# B&R Automation Studio project TD52 (part 87)

#### AI50toIT_mdl.h
```c
/********************************************************************
 * COPYRIGHT -- Bernecker + Rainer Industrie-Elektronik Ges.m.b.H.
 ********************************************************************
 * Program: AI50toIT_mdl
 * File: AI50toIT_mdl.h
 * Author: 105055527
 * Created: Thu Sep 11 18:05:22 2014
 ********************************************************************
 * Header for program AI50toIT_mdl
 ********************************************************************
 * Generated with B&R Automation Studio Target for Simulink V4.2
 * (ERT based)
 ********************************************************************/

#ifndef RTW_HEADER_AI50toIT_mdl_h_
#define RTW_HEADER_AI50toIT_mdl_h_
#ifndef AI50toIT_mdl_COMMON_INCLUDES_
# define AI50toIT_mdl_COMMON_INCLUDES_
#include <math.h>
#include "rtwtypes.h"
#endif                                 /* AI50toIT_mdl_COMMON_INCLUDES_ */

#include "AI50toIT_mdl_types.h"
#include "lAI50toIT.h"

/* Macros for accessing real-time model data structure */
#ifndef rtmGetErrorStatus
# define rtmGetErrorStatus(rtm)        ((void*) 0)
#endif

#ifndef rtmSetErrorStatus
# define rtmSetErrorStatus(rtm, val)   ((void) 0)
#endif

#ifndef rtmGetStopRequested
# define rtmGetStopRequested(rtm)      ((void*) 0)
#endif

#ifndef MIN
#define MIN(a,b)                       ((a) < (b) ? (a) : (b))
#endif

#ifndef MAX
#define MAX(a,b)                       ((a) > (b) ? (a) : (b))
#endif

/* Block signals (auto storage) */

/* Block states (auto storage) for system '<Root>' */

/* External inputs (root inport signals with auto storage) */

/* External outputs (root outports fed by signals with auto storage) */

/* Block signals (auto storage) */
extern BlockIO_AI50toIT_mdl AI50toIT_mdl_B;

/* Block states (auto storage) */
extern D_Work_AI50toIT_mdl AI50toIT_mdl_DWork;

/* External inputs (root inport signals with auto storage) */
extern ExternalInputs_AI50toIT_mdl AI50toIT_mdl_U;

/* External outputs (root outports fed by signals with auto storage) */
extern ExternalOutputs_AI50toIT_mdl AI50toIT_mdl_Y;

/* Model entry point functions */
extern void AI50toIT_mdl_initialize(struct AI50toIT* inst);
extern void AI50toIT_mdl_step(struct AI50toIT* inst);
extern void AI50toIT_mdl_terminate(struct AI50toIT* inst);

/*-
 * The generated code includes comments that allow you to trace directly
 * back to the appropriate location in the model.  The basic format
 * is <system>/block_name, where system is the system number (uniquely
 * assigned by Simulink) and block_name is the name of the block.
 *
 * Use the MATLAB hilite_system command to trace the generated code back
 * to the model.  For example,
 *
 * hilite_system('<S3>')    - opens system 3
 * hilite_system('<S3>/Kp') - opens and selects block Kp which resides in S3
 *
 * Here is the system hierarchy for this model
 *
 * '<Root>' : 'AI50toIT_mdl'
 * '<S1>'   : 'AI50toIT_mdl/AI50 filt'
 * '<S2>'   : 'AI50toIT_mdl/DocBlock'
 * '<S3>'   : 'AI50toIT_mdl/Environment Controller'
 * '<S4>'   : 'AI50toIT_mdl/Environment Controller1'
 * '<S5>'   : 'AI50toIT_mdl/Model Info'
 * '<S6>'   : 'AI50toIT_mdl/PID'
 * '<S7>'   : 'AI50toIT_mdl/Saturation Dynamic'
 * '<S8>'   : 'AI50toIT_mdl/PID/PID Autocoding2'
 * '<S9>'   : 'AI50toIT_mdl/PID/Saturation Dynamic'
 * '<S10>'  : 'AI50toIT_mdl/PID/PID Autocoding2/Dead Zone Dynamic'
 * '<S11>'  : 'AI50toIT_mdl/PID/PID Autocoding2/PID'
 * '<S12>'  : 'AI50toIT_mdl/PID/PID Autocoding2/PID/Clamping circuit'
 * '<S13>'  : 'AI50toIT_mdl/PID/PID Autocoding2/PID/Saturation Dynamic'
 * '<S14>'  : 'AI50toIT_mdl/PID/PID Autocoding2/PID/Clamping circuit/Compare To Constant'
 */
#endif                                 /* RTW_HEADER_AI50toIT_mdl_h_ */
```

#### AI50toIT_mdl_private.h
```c
/********************************************************************
 * COPYRIGHT -- Bernecker + Rainer Industrie-Elektronik Ges.m.b.H.
 ********************************************************************
 * Program: AI50toIT_mdl
 * File: AI50toIT_mdl_private.h
 * Author: 105055527
 * Created: Thu Sep 11 18:05:22 2014
 ********************************************************************
 * Header for program AI50toIT_mdl
 ********************************************************************
 * Generated with B&R Automation Studio Target for Simulink V4.2
 * (ERT based)
 ********************************************************************/

#ifndef RTW_HEADER_AI50toIT_mdl_private_h_
#define RTW_HEADER_AI50toIT_mdl_private_h_
#include "rtwtypes.h"
#include <bur/plctypes.h>
#ifndef __RTWTYPES_H__
#error This file requires rtwtypes.h to be included
#else
#ifdef TMWTYPES_PREVIOUSLY_INCLUDED
#error This file requires rtwtypes.h to be included before tmwtypes.h
#else

/* Check for inclusion of an incorrect version of rtwtypes.h */
#ifndef RTWTYPES_ID_C08S16I32L32N32F1
#error This code was generated with a different "rtwtypes.h" than the file included
#endif                                 /* RTWTYPES_ID_C08S16I32L32N32F1 */
#endif                                 /* TMWTYPES_PREVIOUSLY_INCLUDED */
#endif                                 /* __RTWTYPES_H__ */

#ifndef MIN
#define MIN(a,b)                       ((a) < (b) ? (a) : (b))
#endif

#ifndef MAX
#define MAX(a,b)                       ((a) > (b) ? (a) : (b))
#endif

/* Imported (extern) block parameters */
extern real32_T Kt;                    /* Variable: Kt
                                        * Referenced by: '<S6>/Constant10'
                                        */
extern real32_T N;                     /* Variable: N
                                        * Referenced by: '<S6>/Constant8'
                                        */
extern real32_T T_filt_AI50;           /* Variable: T_filt_AI50
                                        * Referenced by: '<S1>/Constant3'
                                        */
extern real32_T deadband;              /* Variable: deadband
                                        * Referenced by: '<S6>/Constant11'
                                        */
extern real32_T kd;                    /* Variable: kd
                                        * Referenced by: '<S6>/Constant7'
                                        */
extern real32_T ki;                    /* Variable: ki
                                        * Referenced by: '<S6>/Constant6'
                                        */
extern real32_T kp;                    /* Variable: kp
                                        * Referenced by: '<S6>/Constant5'
                                        */
extern real32_T umax;                  /* Variable: umax
                                        * Referenced by: '<S6>/Constant16'
                                        */
extern real32_T umin;                  /* Variable: umin
                                        * Referenced by: '<S6>/Constant17'
                                        */
extern int16_T mode;                   /* Variable: mode
                                        * Referenced by: '<S6>/Constant'
                                        */
extern boolean_T invert;               /* Variable: invert
                                        * Referenced by: '<S6>/Constant4'
                                        */
extern boolean_T reset;                /* Variable: reset
                                        * Referenced by:
                                        *   '<S1>/Constant2'
                                        *   '<S6>/Constant1'
                                        */

#endif                                 /* RTW_HEADER_AI50toIT_mdl_private_h_ */
```

#### AI50toIT_mdl_types.h
```c
/********************************************************************
 * COPYRIGHT -- Bernecker + Rainer Industrie-Elektronik Ges.m.b.H.
 ********************************************************************
 * Program: AI50toIT_mdl
 * File: AI50toIT_mdl_types.h
 * Author: 105055527
 * Created: Thu Sep 11 18:05:22 2014
 ********************************************************************
 * Header for program AI50toIT_mdl
 ********************************************************************
 * Generated with B&R Automation Studio Target for Simulink V4.2
 * (ERT based)
 ********************************************************************/

#ifndef RTW_HEADER_AI50toIT_mdl_types_h_
#define RTW_HEADER_AI50toIT_mdl_types_h_
#ifndef MIN
#define MIN(a,b)                       ((a) < (b) ? (a) : (b))
#endif

#ifndef MAX
#define MAX(a,b)                       ((a) > (b) ? (a) : (b))
#endif
#endif                                 /* RTW_HEADER_AI50toIT_mdl_types_h_ */
```

#### rtwtypes.h
```c
/********************************************************************
 * COPYRIGHT -- Bernecker + Rainer Industrie-Elektronik Ges.m.b.H.
 ********************************************************************
 * Program: AI50toIT_mdl
 * File: rtwtypes.h
 * Author: 105055527
 * Created: Thu Sep 11 18:05:22 2014
 ********************************************************************
 * Header for program AI50toIT_mdl
 ********************************************************************
 * Generated with B&R Automation Studio Target for Simulink V4.2
 * (ERT based)
 ********************************************************************/

#ifndef __RTWTYPES_H__
#define __RTWTYPES_H__
#ifndef TRUE
# define TRUE                          (1U)
#endif

#ifndef FALSE
# define FALSE                         (0U)
#endif

#ifndef __TMWTYPES__
#define __TMWTYPES__
#include <limits.h>

/*=======================================================================*
 * Target hardware information
 *   Device type: Intel->x86/Pentium
 *   Number of bits:     char:   8    short:   16    long:  32
 *                       long:  32
 *                       native word size:  32
 *   Byte ordering: LittleEndian
 *   Signed integer division rounds to: Zero
 *   Shift right on a signed integer as arithmetic shift: on
 *=======================================================================*/

/*=======================================================================*
 * Fixed width word size data types:                                     *
 *   int8_T, int16_T, int32_T     - signed 8, 16, or 32 bit integers     *
 *   uint8_T, uint16_T, uint32_T  - unsigned 8, 16, or 32 bit integers   *
 *   real32_T, real64_T           - 32 and 64 bit floating point numbers *
 *=======================================================================*/
typedef signed char int8_T;
typedef unsigned char uint8_T;
typedef short int16_T;
typedef unsigned short uint16_T;
typedef long int32_T;
typedef unsigned long uint32_T;
typedef float real32_T;
typedef double real64_T;

/*===========================================================================*
 * Generic type definitions: real_T, time_T, boolean_T, int_T, uint_T,       *
 *                           ulong_T, char_T and byte_T.                     *
 *===========================================================================*/
typedef double real_T;
typedef double time_T;
typedef unsigned char boolean_T;
typedef long int_T;
typedef unsigned long uint_T;
typedef unsigned long ulong_T;
typedef char char_T;
typedef unsigned char uchar_T;
typedef char_T byte_T;

/*=======================================================================*
 * Min and Max:                                                          *
 *   int8_T, int16_T, int32_T     - signed 8, 16, or 32 bit integers     *
 *   uint8_T, uint16_T, uint32_T  - unsigned 8, 16, or 32 bit integers   *
 *=======================================================================*/
#define MAX_int8_T                     ((int8_T)(127))
#define MIN_int8_T                     ((int8_T)(-128))
#define MAX_uint8_T                    ((uint8_T)(255U))
#define MIN_uint8_T                    ((uint8_T)(0U))
#define MAX_int16_T                    ((int16_T)(32767))
#define MIN_int16_T                    ((int16_T)(-32768))
#define MAX_uint16_T                   ((uint16_T)(65535U))
#define MIN_uint16_T                   ((uint16_T)(0U))
#define MAX_int32_T                    ((int32_T)(2147483647))
#define MIN_int32_T                    ((int32_T)(-2147483647-1))
#define MAX_uint32_T                   ((uint32_T)(0xFFFFFFFFU))
#define MIN_uint32_T                   ((uint32_T)(0U))

/* Logical type definitions */
#if (!defined(__cplusplus)) && (!defined(__true_false_are_keywords))
#  ifndef false
#   define false                       (0U)
#  endif

#  ifndef true
#   define true                        (1U)
#  endif
#endif

/*
 * Simulink Coder assumes the code is compiled on a target using a 2's complement representation
 * for signed integer values.
 */
#if ((SCHAR_MIN + 1) != -SCHAR_MAX)
#error "This code must be compiled using a 2's complement representation for signed integer values"
#endif

/* This ID is used to detect inclusion of an incompatible rtwtypes.h */
#define RTWTYPES_ID_C08S16I32L32N32F1
#else                                  /* __TMWTYPES__ */
#define TMWTYPES_PREVIOUSLY_INCLUDED
#endif                                 /* __TMWTYPES__ */

/* Block D-Work pointer type */
typedef void * pointer_T;

/* Simulink specific types */
#ifndef __SIMSTRUC_TYPES_H__
#define __SIMSTRUC_TYPES_H__

/* Trigger directions: falling, either, and rising */
typedef enum {
  FALLING_ZERO_CROSSING = -1,
  ANY_ZERO_CROSSING = 0,
  RISING_ZERO_CROSSING = 1
} ZCDirection;

/* Previous state of a trigger signal */
typedef uint8_T ZCSigState;

/* Initial value of a trigger zero crossing signal */
#define UNINITIALIZED_ZCSIG            0x03U
#define NEG_ZCSIG                      0x02U
#define POS_ZCSIG                      0x01U
#define ZERO_ZCSIG                     0x00U

/* Current state of a trigger signal */
typedef enum {
  FALLING_ZCEVENT = -1,
  NO_ZCEVENT = 0,
  RISING_ZCEVENT = 1
} ZCEventType;

#endif                                 /* __SIMSTRUC_TYPES_H__ */
#endif                                 /* __RTWTYPES_H__ */

#ifndef MIN
#define MIN(a,b)                       ((a) < (b) ? (a) : (b))
#endif

#ifndef MAX
#define MAX(a,b)                       ((a) > (b) ? (a) : (b))
#endif
```

#### AI50toIT.c
```c
/********************************************************************
 * COPYRIGHT -- Bernecker + Rainer Industrie-Elektronik Ges.m.b.H.
 ********************************************************************
 * Program: AI50toIT_mdl
 * File: AI50toIT.c
 * Author: 105055527
 * Created: Thu Sep 11 18:05:22 2014
 ********************************************************************
 * Implementation of program AI50toIT_mdl
 ********************************************************************
 * Generated with B&R Automation Studio Target for Simulink V4.2
 * (ERT based)
 ********************************************************************/
#include <bur/plctypes.h>
#include "AI50toIT_mdl.h"
#include "rtwtypes.h"

/* Defines */
#define SS_TERMINATE 4
#define SS_OUTPUT 3
#define SS_INITIALIZE 2

/*  Data Types */

/**************************** GLOBAL DATA *************************************/
/*  Definitions */

/*  Declarations  */

/***************************** FILE SCOPE DATA ********************************/

/*************************** FUNCTIONS ****************************************/
#ifdef __cplusplus

unsigned long bur_heap_size = 6553500;

#endif

void AI50toIT(struct AI50toIT* inst)
{

  switch (inst->ssMethodType)
  {
   case SS_INITIALIZE:
    /* call model initialize function */
    AI50toIT_mdl_initialize(inst);
    break;

   case SS_OUTPUT:
    /* call model step function */
    AI50toIT_mdl_step(inst);

    break;

   case SS_TERMINATE:
    /* call model terminate function */
    AI50toIT_mdl_terminate(inst);
    break;
  }
}

/*****************************************************************************
   Function block sample time: 0.08s
 *****************************************************************************/

/*****************************************************************************
   B&R Automation Studio Target for Simulink Version: A4.5.1 (27-Jul-2015)
 *****************************************************************************/

/*======================== TOOL VERSION INFORMATION ==========================*
 * MATLAB 8.0 (R2012b)20-Jul-2012                                             *
 * Simulink 8.0 (R2012b)20-Jul-2012                                           *
 * Simulink Coder 8.3 (R2012b)20-Jul-2012                                     *
 * Embedded Coder 6.3 (R2012b)20-Jul-2012                                     *
 * Stateflow 8.0 (R2012b)20-Jul-2012                                          *
 *============================================================================*/

/*======================= LICENSE IN USE INFORMATION =========================*
 * matlab                                                                     *
 * matlab_coder                                                               *
 * real-time_workshop                                                         *
 * rtw_embedded_coder                                                         *
 * simulink                                                                   *
 *============================================================================*/
```

#### AI50toIT_mdl.c
```c
/********************************************************************
 * COPYRIGHT -- Bernecker + Rainer Industrie-Elektronik Ges.m.b.H.
 ********************************************************************
 * Program: AI50toIT_mdl
 * File: AI50toIT_mdl.c
 * Author: 105055527
 * Created: Thu Sep 11 18:05:22 2014
 ********************************************************************
 * Implementation of program AI50toIT_mdl
 ********************************************************************
 * Generated with B&R Automation Studio Target for Simulink V4.2
 * (ERT based)
 ********************************************************************/
#include "AI50toIT_mdl.h"
#include "AI50toIT_mdl_private.h"

/*  Defines */

/*  Data Types */

/**************************** GLOBAL DATA *************************************/
/*  Definitions */

/* Block signals (auto storage) */
struct BlockIO_AI50toIT_mdl AI50toIT_mdl_B;

/* Block states (auto storage) */
struct D_Work_AI50toIT_mdl AI50toIT_mdl_DWork;

/* External inputs (root inport signals with auto storage) */
ExternalInputs_AI50toIT_mdl AI50toIT_mdl_U;

/* External outputs (root outports fed by signals with auto storage) */
ExternalOutputs_AI50toIT_mdl AI50toIT_mdl_Y;

/*  Declarations  */

/***************************** FILE SCOPE DATA ********************************/

/*************************** FUNCTIONS ****************************************/

/* Model step function */
void AI50toIT_mdl_step(struct AI50toIT* inst)
{
  real32_T rtb_Add[25];
  real32_T rtb_Abs[25];
  real32_T rtb_Trackingswitch;
  real32_T rtb_Invertswitch;
  real32_T rtb_SumI1[25];
  boolean_T rtb_LowerRelop1_k[25];
  int32_T i;
  real32_T rtb_SumI;
  real32_T rtb_SumI_0;

  /* S-Function (bur_in): '<Root>/Input16' */
  {
    int_T i1;
    real32_T *y0 = AI50toIT_mdl_B.Input16;
    for (i1=0; i1 < 25; i1++) {
      y0[i1] = inst->uman[i1];
    }
  }

  /* Switch: '<S8>/Invert switch' incorporates:
   *  Constant: '<S6>/Constant4'
   *  Constant: '<S8>/Constant2'
   *  Constant: '<S8>/Constant3'
   */
  if ((int32_T)inst->invert > 0) {
    rtb_Invertswitch = -1.0F;
  } else {
    rtb_Invertswitch = 1.0F;
  }

  /* End of Switch: '<S8>/Invert switch' */

  /* S-Function (bur_in): '<Root>/Input5' */
  AI50toIT_mdl_B.Input5 = inst->AI50ref;

  /* S-Function (bur_in): '<Root>/Input8' */
  {
    int_T i1;
    real32_T *y0 = AI50toIT_mdl_B.Input8;
    for (i1=0; i1 < 25; i1++) {
      y0[i1] = inst->AI50offset[i1];
    }
  }

  /* S-Function (bur_in): '<Root>/Input3' */
  {
    int_T i1;
    real32_T *y0 = AI50toIT_mdl_B.Input3;
    for (i1=0; i1 < 25; i1++) {
      y0[i1] = inst->AI50offset_knck[i1];
    }
  }

  /* S-Function (bur_in): '<Root>/Input4' */
  AI50toIT_mdl_B.Input4 = inst->K_knck;

  /* Sum: '<Root>/Add' incorporates:
   *  Product: '<Root>/Product'
   */
  for (i = 0; i < 25; i++) {
    rtb_Add[i] = (AI50toIT_mdl_B.Input5 + AI50toIT_mdl_B.Input8[i]) +
      AI50toIT_mdl_B.Input3[i] * AI50toIT_mdl_B.Input4;
  }

  /* End of Sum: '<Root>/Add' */

  /* DiscreteIntegrator: '<S1>/Discrete-Time Integrator' incorporates:
   *  Constant: '<S1>/Constant2'
   */
  if (inst->reset || (AI50toIT_mdl_DWork.DiscreteTimeIntegrator_PrevRese != 0)) {
    for (i = 0; i < 25; i++) {
      AI50toIT_mdl_DWork.DiscreteTimeIntegrator_DSTATE[i] = 10.0F;
    }
  }

  for (i = 0; i < 25; i++) {
    /* DiscreteIntegrator: '<S1>/Discrete-Time Integrator' */
    AI50toIT_mdl_B.DiscreteTimeIntegrator[i] =
      AI50toIT_mdl_DWork.DiscreteTimeIntegrator_DSTATE[i];

    /* Sum: '<S8>/Sum' incorporates:
     *  Product: '<S8>/Product'
     *  Product: '<S8>/Product1'
     */
    rtb_Trackingswitch = rtb_Add[i] - AI50toIT_mdl_B.DiscreteTimeIntegrator[i];

    /* Switch: '<S10>/Switch' incorporates:
     *  Constant: '<S6>/Constant11'
     *  Gain: '<S8>/Gain1'
     *  RelationalOperator: '<S10>/u_GTE_up'
     *  RelationalOperator: '<S10>/u_GT_lo'
     *  Switch: '<S10>/Switch1'
     */
    if (rtb_Trackingswitch >= inst->deadband) {
      rtb_SumI = inst->deadband;
    } else if (rtb_Trackingswitch > -inst->deadband) {
      /* Switch: '<S10>/Switch1' */
      rtb_SumI = rtb_Trackingswitch;
    } else {
      rtb_SumI = -inst->deadband;
    }

    /* End of Switch: '<S10>/Switch' */

    /* Product: '<S8>/Product2' incorporates:
     *  Sum: '<S10>/Diff'
     */
    AI50toIT_mdl_B.Product2[i] = (rtb_Trackingswitch - rtb_SumI) *
      rtb_Invertswitch;

    /* Product: '<S11>/Product1' incorporates:
     *  Constant: '<S6>/Constant5'
     */
    AI50toIT_mdl_B.Product1[i] = inst->kp * AI50toIT_mdl_B.Product2[i];

    /* Sum: '<S8>/Sum' */
    rtb_Abs[i] = rtb_Trackingswitch;
  }

  for (i = 0; i < 25; i++) {
    /* DiscreteIntegrator: '<S11>/Integrator' incorporates:
     *  Constant: '<S6>/Constant1'
     */
    if (inst->reset) {
      AI50toIT_mdl_DWork.Integrator_DSTATE[i] = 0.0F;
    }

    AI50toIT_mdl_B.Integrator[i] = AI50toIT_mdl_DWork.Integrator_DSTATE[i];

    /* End of DiscreteIntegrator: '<S11>/Integrator' */

    /* DiscreteIntegrator: '<S11>/Filter' incorporates:
     *  Constant: '<S6>/Constant1'
     */
    if (inst->reset) {
      AI50toIT_mdl_DWork.Filter_DSTATE[i] = 0.0F;
    }

    /* Product: '<S11>/Product4' incorporates:
     *  Constant: '<S6>/Constant7'
     *  Constant: '<S6>/Constant8'
     *  DiscreteIntegrator: '<S11>/Filter'
     *  Product: '<S11>/Product3'
     *  Sum: '<S11>/SumD'
     */
    AI50toIT_mdl_B.Product4[i] = (AI50toIT_mdl_B.Product2[i] * inst->kd -
      AI50toIT_mdl_DWork.Filter_DSTATE[i]) * inst->N;

    /* Sum: '<S11>/Sum2' incorporates:
     *  Sum: '<S11>/Sum1'
     */
    rtb_SumI = (AI50toIT_mdl_B.Product1[i] + AI50toIT_mdl_B.Integrator[i]) +
      AI50toIT_mdl_B.Product4[i];

    /* Switch: '<S13>/Switch2' incorporates:
     *  Constant: '<S6>/Constant12'
     *  Constant: '<S6>/Constant14'
     *  RelationalOperator: '<S13>/LowerRelop1'
     *  RelationalOperator: '<S13>/UpperRelop'
     *  Switch: '<S13>/Switch'
     */
    if (rtb_SumI > 20.0F) {
      AI50toIT_mdl_B.Switch2[i] = 20.0F;
    } else if (rtb_SumI < -20.0F) {
      /* Switch: '<S13>/Switch' incorporates:
       *  Constant: '<S6>/Constant14'
       */
      AI50toIT_mdl_B.Switch2[i] = -20.0F;
    } else {
      AI50toIT_mdl_B.Switch2[i] = rtb_SumI;
    }

    /* End of Switch: '<S13>/Switch2' */

    /* Sum: '<S11>/Sum2' */
    rtb_SumI1[i] = rtb_SumI;
  }

  /* MultiPortSwitch: '<S8>/Mode switch' incorporates:
   *  Constant: '<S6>/Constant'
   */
  switch (inst->mode) {
   case 1:
    for (i = 0; i < 25; i++) {
      AI50toIT_mdl_B.Modeswitch[i] = AI50toIT_mdl_B.Input16[i];
    }
    break;

   case 2:
    for (i = 0; i < 25; i++) {
      AI50toIT_mdl_B.Modeswitch[i] = AI50toIT_mdl_B.Input16[i];
    }
    break;

   default:
    for (i = 0; i < 25; i++) {
      AI50toIT_mdl_B.Modeswitch[i] = AI50toIT_mdl_B.Switch2[i];
    }
    break;
  }

  for (i = 0; i < 25; i++) {
    /* Switch: '<S9>/Switch2' incorporates:
     *  Constant: '<S6>/Constant16'
     *  Constant: '<S6>/Constant17'
     *  RelationalOperator: '<S9>/LowerRelop1'
     *  RelationalOperator: '<S9>/UpperRelop'
     *  Switch: '<S9>/Switch'
     */
    if (AI50toIT_mdl_B.Modeswitch[i] > inst->umax) {
      /* Outport: '<Root>/IToffset' */
      AI50toIT_mdl_Y.IToffset[i] = inst->umax;
    } else if (AI50toIT_mdl_B.Modeswitch[i] < inst->umin) {
      /* Switch: '<S9>/Switch' incorporates:
       *  Constant: '<S6>/Constant17'
       *  Outport: '<Root>/IToffset'
       */
      AI50toIT_mdl_Y.IToffset[i] = inst->umin;
    } else {
      /* Outport: '<Root>/IToffset' incorporates:
       *  Switch: '<S9>/Switch'
       */
      AI50toIT_mdl_Y.IToffset[i] = AI50toIT_mdl_B.Modeswitch[i];
    }

    /* End of Switch: '<S9>/Switch2' */

    /* Outport: '<Root>/ITsat' incorporates:
     *  Sum: '<S6>/Sum2'
     */
    AI50toIT_mdl_Y.ITsat[i] = AI50toIT_mdl_Y.IToffset[i] -
      AI50toIT_mdl_B.Modeswitch[i];

    /* Outport: '<Root>/AI50err' incorporates:
     *  Sum: '<S6>/Sum3'
     */
    AI50toIT_mdl_Y.AI50err[i] = rtb_Add[i] -
      AI50toIT_mdl_B.DiscreteTimeIntegrator[i];
  }

  /* End of MultiPortSwitch: '<S8>/Mode switch' */

  /* S-Function (bur_out): '<Root>/Output1' */
  {
    int_T i1;
    const real32_T *u0 = &AI50toIT_mdl_Y.ITsat[0];
    for (i1=0; i1 < 25; i1++) {
      inst->ITsat[i1] = u0[i1];
    }
  }

  /* S-Function (bur_out): '<Root>/Output2' */
  {
    int_T i1;
    const real32_T *u0 = &AI50toIT_mdl_Y.AI50err[0];
    for (i1=0; i1 < 25; i1++) {
      inst->AI50err[i1] = u0[i1];
    }
  }

  /* S-Function (bur_out): '<Root>/Output3' */
  {
    int_T i1;
    const real32_T *u0 = &AI50toIT_mdl_Y.IToffset[0];
    for (i1=0; i1 < 25; i1++) {
      inst->IToffset[i1] = u0[i1];
    }
  }

  /* S-Function (bur_out): '<Root>/Output6' */
  {
    int_T i1;
    const real32_T *u0 = AI50toIT_mdl_B.DiscreteTimeIntegrator;
    for (i1=0; i1 < 25; i1++) {
      inst->DB_AI50_f[i1] = u0[i1];
    }
  }

  /* S-Function (bur_in): '<Root>/Input1' */
  AI50toIT_mdl_B.Input1 = inst->AI50_max;

  /* S-Function (bur_in): '<Root>/Input9' */
  {
    int_T i1;
    real32_T *y0 = AI50toIT_mdl_B.Input9;
    for (i1=0; i1 < 25; i1++) {
      y0[i1] = inst->AI50act[i1];
    }
  }

  /* RelationalOperator: '<S7>/LowerRelop1' */
  for (i = 0; i < 25; i++) {
    rtb_LowerRelop1_k[i] = (AI50toIT_mdl_B.Input9[i] > AI50toIT_mdl_B.Input1);
  }

  /* End of RelationalOperator: '<S7>/LowerRelop1' */

  /* S-Function (bur_in): '<Root>/Input2' */
  AI50toIT_mdl_B.Input2 = inst->AI50_min;

  /* Sum: '<S1>/Sum2' */
  for (i = 0; i < 25; i++) {
    /* Switch: '<S7>/Switch2' incorporates:
     *  RelationalOperator: '<S7>/UpperRelop'
     *  Switch: '<S7>/Switch'
     */
    if (rtb_LowerRelop1_k[i]) {
      rtb_Trackingswitch = AI50toIT_mdl_B.Input1;
    } else if (AI50toIT_mdl_B.Input9[i] < AI50toIT_mdl_B.Input2) {
      /* Switch: '<S7>/Switch' */
      rtb_Trackingswitch = AI50toIT_mdl_B.Input2;
    } else {
      rtb_Trackingswitch = AI50toIT_mdl_B.Input9[i];
    }

    /* End of Switch: '<S7>/Switch2' */
    rtb_Abs[i] = rtb_Trackingswitch - AI50toIT_mdl_B.DiscreteTimeIntegrator[i];
  }

  /* End of Sum: '<S1>/Sum2' */

  /* Saturate: '<S1>/Saturation' incorporates:
   *  Constant: '<S1>/Constant3'
   */
  if (inst->T_filt_AI50 >= 0.001F) {
    rtb_Invertswitch = inst->T_filt_AI50;
  } else {
    rtb_Invertswitch = 0.001F;
  }

  /* End of Saturate: '<S1>/Saturation' */

  /* S-Function (bur_out): '<S6>/Output5' */
  inst->dbg1[0] = AI50toIT_mdl_B.Modeswitch[1];
  inst->dbg1[1] = AI50toIT_mdl_B.Switch2[1];
  inst->dbg1[2] = AI50toIT_mdl_B.Product1[1];
  inst->dbg1[3] = AI50toIT_mdl_B.Integrator[1];
  inst->dbg1[4] = AI50toIT_mdl_B.Product4[1];
  inst->dbg1[5] = AI50toIT_mdl_B.Product2[1];
  for (i = 0; i < 25; i++) {
    /* Sum: '<S12>/Sum' incorporates:
     *  Signum: '<S12>/SignPreSat'
     */
    rtb_SumI = AI50toIT_mdl_Y.IToffset[i] - rtb_SumI1[i];

    /* RelationalOperator: '<S14>/Compare' incorporates:
     *  Abs: '<S12>/Abs'
     *  Constant: '<S14>/Constant'
     */
    rtb_LowerRelop1_k[i] = ((real32_T)fabs(rtb_SumI) > 0.1F);

    /* Signum: '<S12>/SignPreSat' */
    if (rtb_SumI < 0.0F) {
      rtb_Add[i] = -1.0F;
    } else if (rtb_SumI > 0.0F) {
      rtb_Add[i] = 1.0F;
    } else {
      rtb_Add[i] = rtb_SumI;
    }
  }

  /* MultiPortSwitch: '<S8>/Tracking switch' incorporates:
   *  Constant: '<S6>/Constant'
   *  Constant: '<S6>/Constant10'
   *  Constant: '<S8>/Constant1'
   */
  switch (inst->mode) {
   case 1:
    rtb_Trackingswitch = 0.0F;
    break;

   case 2:
    rtb_Trackingswitch = inst->Kt;
    break;

   default:
    rtb_Trackingswitch = 0.0F;
    break;
  }

  for (i = 0; i < 25; i++) {
    /* Sum: '<S11>/SumI1' incorporates:
     *  Constant: '<S6>/Constant6'
     *  Product: '<S11>/Product'
     *  Product: '<S11>/Product2'
     *  Sum: '<S11>/SumI3'
     */
    rtb_SumI = (AI50toIT_mdl_B.Input16[i] - AI50toIT_mdl_B.Switch2[i]) *
      rtb_Trackingswitch + AI50toIT_mdl_B.Product2[i] * inst->ki;

    /* Switch: '<S11>/Switch' incorporates:
     *  Constant: '<S11>/Constant4'
     *  Logic: '<S12>/AND'
     *  RelationalOperator: '<S12>/Equal'
     */
    if (rtb_SumI < 0.0F) {
      rtb_SumI_0 = -1.0F;
    } else if (rtb_SumI > 0.0F) {
      rtb_SumI_0 = 1.0F;
    } else {
      rtb_SumI_0 = rtb_SumI;
    }

    if (rtb_LowerRelop1_k[i] && (rtb_Add[i] != rtb_SumI_0)) {
      rtb_SumI = 0.0F;
    }

    rtb_Add[i] = rtb_SumI;

    /* End of Switch: '<S11>/Switch' */
  }

  /* End of MultiPortSwitch: '<S8>/Tracking switch' */

  /* Update for DiscreteIntegrator: '<S1>/Discrete-Time Integrator' incorporates:
   *  Constant: '<S1>/Constant2'
   *  Product: '<S1>/Divide'
   */
  if (inst->reset == 0) {
    for (i = 0; i < 25; i++) {
      AI50toIT_mdl_DWork.DiscreteTimeIntegrator_DSTATE[i] += rtb_Abs[i] /
        rtb_Invertswitch * 0.08F;
    }
  }

  if ((int32_T)inst->reset > 0) {
    AI50toIT_mdl_DWork.DiscreteTimeIntegrator_PrevRese = 1;
  } else if (inst->reset == 0) {
    AI50toIT_mdl_DWork.DiscreteTimeIntegrator_PrevRese = 0;
  } else {
    AI50toIT_mdl_DWork.DiscreteTimeIntegrator_PrevRese = 2;
  }

  for (i = 0; i < 25; i++) {
    /* Update for DiscreteIntegrator: '<S11>/Integrator' */
    AI50toIT_mdl_DWork.Integrator_DSTATE[i] += 0.08F * rtb_Add[i];

    /* Update for DiscreteIntegrator: '<S11>/Filter' */
    AI50toIT_mdl_DWork.Filter_DSTATE[i] += 0.08F * AI50toIT_mdl_B.Product4[i];
  }

  /* End of Update for DiscreteIntegrator: '<S1>/Discrete-Time Integrator' */
}

/* Model initialize function */
void AI50toIT_mdl_initialize(struct AI50toIT* inst)
{
  /* S-Function (bur_out): '<Root>/Output7' */
  inst->DB_Ts = 0.08;

  {
    int32_T i;
    for (i = 0; i < 25; i++) {
      /* InitializeConditions for DiscreteIntegrator: '<S1>/Discrete-Time Integrator' */
      AI50toIT_mdl_DWork.DiscreteTimeIntegrator_DSTATE[i] = 10.0F;
    }
  }
}

/* Model terminate function */
void AI50toIT_mdl_terminate(struct AI50toIT* inst)
{
  /* (no terminate code required) */
}

/*======================== TOOL VERSION INFORMATION ==========================*
 * MATLAB 8.0 (R2012b)20-Jul-2012                                             *
 * Simulink 8.0 (R2012b)20-Jul-2012                                           *
 * Simulink Coder 8.3 (R2012b)20-Jul-2012                                     *
 * Embedded Coder 6.3 (R2012b)20-Jul-2012                                     *
 * Stateflow 8.0 (R2012b)20-Jul-2012                                          *
 *============================================================================*/

/*======================= LICENSE IN USE INFORMATION =========================*
 * matlab                                                                     *
 * matlab_coder                                                               *
 * real-time_workshop                                                         *
 * rtw_embedded_coder                                                         *
 * simulink                                                                   *
 *============================================================================*/
```

#### lib_properties.txt
```
For manual assignment to hardware configuration please
add the following additional include directories:

\Logical\MATLAB_includes\R2012b\

And the following additional build options:

-lm -D MODEL=AI50toIT_mdl -D NUMST=1 -D NCSTATES=0 -D HAVESTDIO -D ONESTEPFCN=1 -D TERMFCN=1 -D MAT_FILE=0 -D MULTI_INSTANCE_CODE=0 -D INTEGER_CODE=0 -D MT=0 -D CLASSIC_INTERFACE=0 -D TID01EQ=0
```

### Library Logical/EngineController/Sondergas/lCoV (ANSIC)

#### lCoV.fun
```iecst
FUNCTION_BLOCK CoV
  VAR_INPUT
    ssMethodType: SINT;
  END_VAR  VAR_OUTPUT
        CoV : ARRAY[0..24] OF REAL; (**)
  END_VAR
  VAR_OUTPUT
        Avg : ARRAY[0..24] OF REAL; (**)
  END_VAR
  VAR_OUTPUT
        Std : ARRAY[0..24] OF REAL; (**)
  END_VAR
  VAR_INPUT
        In : ARRAY[0..24] OF REAL; (**)
  END_VAR
	VAR
		bur_BlockIO_CoV_24Cyl : BlockIO_CoV_24Cyl;
	END_VAR
	VAR
		bur_D_Work_CoV_24Cyl : D_Work_CoV_24Cyl;
	END_VAR
END_FUNCTION_BLOCK
```

#### lCoV.typ
```iecst
TYPE

END_TYPE
TYPE
BlockIO_CoV_24Cyl : STRUCT
	Avg : REAL;
	Std : REAL;
	CoV : REAL;
	Avg_g : REAL;
	Std_n : REAL;
	CoV_c : REAL;
	Avg_d : REAL;
	Std_f : REAL;
	CoV_d : REAL;
	Avg_m : REAL;
	Std_i : REAL;
	CoV_m : REAL;
	Avg_dg : REAL;
	Std_g : REAL;
	CoV_k : REAL;
	Avg_h : REAL;
	Std_h : REAL;
	CoV_e : REAL;
	Avg_c : REAL;
	Std_k : REAL;
	CoV_mz : REAL;
	Avg_a : REAL;
	Std_kl : REAL;
	CoV_db : REAL;
	Avg_n : REAL;
	Std_j : REAL;
	CoV_n : REAL;
	Avg_n5 : REAL;
	Std_gz : REAL;
	CoV_l : REAL;
	Avg_m0 : REAL;
	Std_l : REAL;
	CoV_cl : REAL;
	Avg_e : REAL;
	Std_hh : REAL;
	CoV_me : REAL;
	Avg_n4 : REAL;
	Std_hx : REAL;
	CoV_lo : REAL;
	Avg_e5 : REAL;
	Std_e : REAL;
	CoV_f : REAL;
	Avg_eu : REAL;
	Std_m : REAL;
	CoV_i : REAL;
	Avg_ey : REAL;
	Std_b : REAL;
	CoV_lh : REAL;
	Avg_j : REAL;
	Std_ev : REAL;
	CoV_mw : REAL;
	Avg_p : REAL;
	Std_a : REAL;
	CoV_iy : REAL;
	Avg_gz : REAL;
	Std_d : REAL;
	CoV_cc : REAL;
	Avg_pv : REAL;
	Std_ht : REAL;
	CoV_h : REAL;
	Avg_d2 : REAL;
	Std_ji : REAL;
	CoV_hj : REAL;
	Avg_b : REAL;
	Std_ag : REAL;
	CoV_j : REAL;
	Avg_o : REAL;
	Std_gd : REAL;
	CoV_nw : REAL;
	Avg_l : REAL;
	Std_ik : REAL;
	CoV_o : REAL;
	Avg_lu : REAL;
	Std_c : REAL;
	CoV_ja : REAL;
	Input25 : ARRAY[0..24] OF REAL;
	Selector : REAL;
	Selector_l : REAL;
	Selector_a : REAL;
	Selector_n : REAL;
	Selector_c : REAL;
	Selector_c4 : REAL;
	Selector_g : REAL;
	Selector_o : REAL;
	Selector_ct : REAL;
	Selector_h : REAL;
	Selector_lk : REAL;
	Selector_b : REAL;
	Selector_al : REAL;
	Selector_j : REAL;
	Selector_d : REAL;
	Selector_f : REAL;
	Selector_p : REAL;
	Selector_hu : REAL;
	Selector_ob : REAL;
	Selector_ox : REAL;
	Selector_m : REAL;
	Selector_p5 : REAL;
	Selector_k : REAL;
	Selector_og : REAL;
	Selector_fv : REAL;
END_STRUCT;
D_Work_CoV_24Cyl : STRUCT
	TappedDelaysetasN_cyc_X : ARRAY[0..99] OF REAL;
	TappedDelaysetasN_cyc_X_c : ARRAY[0..99] OF REAL;
	TappedDelaysetasN_cyc_X_a : ARRAY[0..99] OF REAL;
	TappedDelaysetasN_cyc_X_ch : ARRAY[0..99] OF REAL;
	TappedDelaysetasN_cyc_X_m : ARRAY[0..99] OF REAL;
	TappedDelaysetasN_cyc_X_b : ARRAY[0..99] OF REAL;
	TappedDelaysetasN_cyc_X_m3 : ARRAY[0..99] OF REAL;
	TappedDelaysetasN_cyc_X_ap : ARRAY[0..99] OF REAL;
	TappedDelaysetasN_cyc_X_d : ARRAY[0..99] OF REAL;
	TappedDelaysetasN_cyc_X_j : ARRAY[0..99] OF REAL;
	TappedDelaysetasN_cyc_X_b0 : ARRAY[0..99] OF REAL;
	TappedDelaysetasN_cyc_X_da : ARRAY[0..99] OF REAL;
	TappedDelaysetasN_cyc_X_di : ARRAY[0..99] OF REAL;
	TappedDelaysetasN_cyc_X_g : ARRAY[0..99] OF REAL;
	TappedDelaysetasN_cyc_X_jg : ARRAY[0..99] OF REAL;
	TappedDelaysetasN_cyc_X_l : ARRAY[0..99] OF REAL;
	TappedDelaysetasN_cyc_X_f : ARRAY[0..99] OF REAL;
	TappedDelaysetasN_cyc_X_n : ARRAY[0..99] OF REAL;
	TappedDelaysetasN_cyc_X_f0 : ARRAY[0..99] OF REAL;
	TappedDelaysetasN_cyc_X_ln : ARRAY[0..99] OF REAL;
	TappedDelaysetasN_cyc_X_jc : ARRAY[0..99] OF REAL;
	TappedDelaysetasN_cyc_X_i : ARRAY[0..99] OF REAL;
	TappedDelaysetasN_cyc_X_mr : ARRAY[0..99] OF REAL;
	TappedDelaysetasN_cyc_X_g1 : ARRAY[0..99] OF REAL;
	TappedDelaysetasN_cyc_X_cc : ARRAY[0..99] OF REAL;
END_STRUCT;
END_TYPE
```

#### CoV_24Cyl.h
```c
/********************************************************************
 * COPYRIGHT -- Bernecker + Rainer Industrie-Elektronik Ges.m.b.H.
 ********************************************************************
 * Program: CoV_24Cyl
 * File: CoV_24Cyl.h
 * Author: 105055527
 * Created: Tue Sep 23 05:31:36 2014
 ********************************************************************
 * Header for program CoV_24Cyl
 ********************************************************************
 * Generated with B&R Automation Studio Target for Simulink V4.2
 * (ERT based)
 ********************************************************************/

#ifndef RTW_HEADER_CoV_24Cyl_h_
#define RTW_HEADER_CoV_24Cyl_h_
#ifndef CoV_24Cyl_COMMON_INCLUDES_
# define CoV_24Cyl_COMMON_INCLUDES_
#include <math.h>
#include "rtwtypes.h"
#endif                                 /* CoV_24Cyl_COMMON_INCLUDES_ */

#include "CoV_24Cyl_types.h"
#include "lCoV.h"

/* Macros for accessing real-time model data structure */
#ifndef rtmGetErrorStatus
# define rtmGetErrorStatus(rtm)        ((void*) 0)
#endif

#ifndef rtmSetErrorStatus
# define rtmSetErrorStatus(rtm, val)   ((void) 0)
#endif

#ifndef rtmGetStopRequested
# define rtmGetStopRequested(rtm)      ((void*) 0)
#endif

#ifndef MIN
#define MIN(a,b)                       ((a) < (b) ? (a) : (b))
#endif

#ifndef MAX
#define MAX(a,b)                       ((a) > (b) ? (a) : (b))
#endif

/* Block signals (auto storage) */

/* Block states (auto storage) for system '<Root>' */

/* Block signals (auto storage) */
extern BlockIO_CoV_24Cyl CoV_24Cyl_B;

/* Block states (auto storage) */
extern D_Work_CoV_24Cyl CoV_24Cyl_DWork;

/* Model entry point functions */
extern void CoV_24Cyl_initialize(struct CoV* inst);
extern void CoV_24Cyl_step(struct CoV* inst);
extern void CoV_24Cyl_terminate(struct CoV* inst);

/*-
 * The generated code includes comments that allow you to trace directly
 * back to the appropriate location in the model.  The basic format
 * is <system>/block_name, where system is the system number (uniquely
 * assigned by Simulink) and block_name is the name of the block.
 *
 * Use the MATLAB hilite_system command to trace the generated code back
 * to the model.  For example,
 *
 * hilite_system('<S3>')    - opens system 3
 * hilite_system('<S3>/Kp') - opens and selects block Kp which resides in S3
 *
 * Here is the system hierarchy for this model
 *
 * '<Root>' : 'CoV_24Cyl'
 * '<S1>'   : 'CoV_24Cyl/CoV_0'
 * '<S2>'   : 'CoV_24Cyl/CoV_1'
 * '<S3>'   : 'CoV_24Cyl/CoV_10'
 * '<S4>'   : 'CoV_24Cyl/CoV_11'
 * '<S5>'   : 'CoV_24Cyl/CoV_12'
 * '<S6>'   : 'CoV_24Cyl/CoV_13'
 * '<S7>'   : 'CoV_24Cyl/CoV_14'
 * '<S8>'   : 'CoV_24Cyl/CoV_15'
 * '<S9>'   : 'CoV_24Cyl/CoV_16'
 * '<S10>'  : 'CoV_24Cyl/CoV_17'
 * '<S11>'  : 'CoV_24Cyl/CoV_18'
 * '<S12>'  : 'CoV_24Cyl/CoV_19'
 * '<S13>'  : 'CoV_24Cyl/CoV_2'
 * '<S14>'  : 'CoV_24Cyl/CoV_20'
 * '<S15>'  : 'CoV_24Cyl/CoV_21'
 * '<S16>'  : 'CoV_24Cyl/CoV_22'
 * '<S17>'  : 'CoV_24Cyl/CoV_23'
 * '<S18>'  : 'CoV_24Cyl/CoV_24'
 * '<S19>'  : 'CoV_24Cyl/CoV_3'
 * '<S20>'  : 'CoV_24Cyl/CoV_4'
 * '<S21>'  : 'CoV_24Cyl/CoV_5'
 * '<S22>'  : 'CoV_24Cyl/CoV_6'
 * '<S23>'  : 'CoV_24Cyl/CoV_7'
 * '<S24>'  : 'CoV_24Cyl/CoV_8'
 * '<S25>'  : 'CoV_24Cyl/CoV_9'
 */
#endif                                 /* RTW_HEADER_CoV_24Cyl_h_ */
```

#### CoV_24Cyl_private.h
```c
/********************************************************************
 * COPYRIGHT -- Bernecker + Rainer Industrie-Elektronik Ges.m.b.H.
 ********************************************************************
 * Program: CoV_24Cyl
 * File: CoV_24Cyl_private.h
 * Author: 105055527
 * Created: Tue Sep 23 05:31:36 2014
 ********************************************************************
 * Header for program CoV_24Cyl
 ********************************************************************
 * Generated with B&R Automation Studio Target for Simulink V4.2
 * (ERT based)
 ********************************************************************/

#ifndef RTW_HEADER_CoV_24Cyl_private_h_
#define RTW_HEADER_CoV_24Cyl_private_h_
#include "rtwtypes.h"
#include <bur/plctypes.h>
#ifndef __RTWTYPES_H__
#error This file requires rtwtypes.h to be included
#else
#ifdef TMWTYPES_PREVIOUSLY_INCLUDED
#error This file requires rtwtypes.h to be included before tmwtypes.h
#else

/* Check for inclusion of an incorrect version of rtwtypes.h */
#ifndef RTWTYPES_ID_C08S16I32L32N32F1
#error This code was generated with a different "rtwtypes.h" than the file included
#endif                                 /* RTWTYPES_ID_C08S16I32L32N32F1 */
#endif                                 /* TMWTYPES_PREVIOUSLY_INCLUDED */
#endif                                 /* __RTWTYPES_H__ */

#ifndef MIN
#define MIN(a,b)                       ((a) < (b) ? (a) : (b))
#endif

#ifndef MAX
#define MAX(a,b)                       ((a) > (b) ? (a) : (b))
#endif
#endif                                 /* RTW_HEADER_CoV_24Cyl_private_h_ */
```

#### CoV_24Cyl_types.h
```c
/********************************************************************
 * COPYRIGHT -- Bernecker + Rainer Industrie-Elektronik Ges.m.b.H.
 ********************************************************************
 * Program: CoV_24Cyl
 * File: CoV_24Cyl_types.h
 * Author: 105055527
 * Created: Tue Sep 23 05:31:36 2014
 ********************************************************************
 * Header for program CoV_24Cyl
 ********************************************************************
 * Generated with B&R Automation Studio Target for Simulink V4.2
 * (ERT based)
 ********************************************************************/

#ifndef RTW_HEADER_CoV_24Cyl_types_h_
#define RTW_HEADER_CoV_24Cyl_types_h_
#ifndef MIN
#define MIN(a,b)                       ((a) < (b) ? (a) : (b))
#endif

#ifndef MAX
#define MAX(a,b)                       ((a) > (b) ? (a) : (b))
#endif
#endif                                 /* RTW_HEADER_CoV_24Cyl_types_h_ */
```

#### rtwtypes.h
```c
/********************************************************************
 * COPYRIGHT -- Bernecker + Rainer Industrie-Elektronik Ges.m.b.H.
 ********************************************************************
 * Program: CoV_24Cyl
 * File: rtwtypes.h
 * Author: 105055527
 * Created: Tue Sep 23 05:31:36 2014
 ********************************************************************
 * Header for program CoV_24Cyl
 ********************************************************************
 * Generated with B&R Automation Studio Target for Simulink V4.2
 * (ERT based)
 ********************************************************************/

#ifndef __RTWTYPES_H__
#define __RTWTYPES_H__
#ifndef TRUE
# define TRUE                          (1U)
#endif

#ifndef FALSE
# define FALSE                         (0U)
#endif

#ifndef __TMWTYPES__
#define __TMWTYPES__
#include <limits.h>

/*=======================================================================*
 * Target hardware information
 *   Device type: Intel->x86/Pentium
 *   Number of bits:     char:   8    short:   16    int:  32
 *                       long:  32
 *                       native word size:  32
 *   Byte ordering: LittleEndian
 *   Signed integer division rounds to: Zero
 *   Shift right on a signed integer as arithmetic shift: on
 *=======================================================================*/

/*=======================================================================*
 * Fixed width word size data types:                                     *
 *   int8_T, int16_T, int32_T     - signed 8, 16, or 32 bit integers     *
 *   uint8_T, uint16_T, uint32_T  - unsigned 8, 16, or 32 bit integers   *
 *   real32_T, real64_T           - 32 and 64 bit floating point numbers *
 *=======================================================================*/
typedef signed char int8_T;
typedef unsigned char uint8_T;
typedef short int16_T;
typedef unsigned short uint16_T;
typedef int int32_T;
typedef unsigned int uint32_T;
typedef float real32_T;
typedef double real64_T;

/*===========================================================================*
 * Generic type definitions: real_T, time_T, boolean_T, int_T, uint_T,       *
 *                           ulong_T, char_T and byte_T.                     *
 *===========================================================================*/
typedef double real_T;
typedef double time_T;
typedef unsigned char boolean_T;
typedef long int int_T;
typedef unsigned int uint_T;
typedef unsigned long ulong_T;
typedef char char_T;
typedef unsigned char uchar_T;
typedef char_T byte_T;

/*=======================================================================*
 * Min and Max:                                                          *
 *   int8_T, int16_T, int32_T     - signed 8, 16, or 32 bit integers     *
 *   uint8_T, uint16_T, uint32_T  - unsigned 8, 16, or 32 bit integers   *
 *=======================================================================*/
#define MAX_int8_T                     ((int8_T)(127))
#define MIN_int8_T                     ((int8_T)(-128))
#define MAX_uint8_T                    ((uint8_T)(255U))
#define MIN_uint8_T                    ((uint8_T)(0U))
#define MAX_int16_T                    ((int16_T)(32767))
#define MIN_int16_T                    ((int16_T)(-32768))
#define MAX_uint16_T                   ((uint16_T)(65535U))
#define MIN_uint16_T                   ((uint16_T)(0U))
#define MAX_int32_T                    ((int32_T)(2147483647))
#define MIN_int32_T                    ((int32_T)(-2147483647-1))
#define MAX_uint32_T                   ((uint32_T)(0xFFFFFFFFU))
#define MIN_uint32_T                   ((uint32_T)(0U))

/* Logical type definitions */
#if (!defined(__cplusplus)) && (!defined(__true_false_are_keywords))
#  ifndef false
#   define false                       (0U)
#  endif

#  ifndef true
#   define true                        (1U)
#  endif
#endif

/*
 * Simulink Coder assumes the code is compiled on a target using a 2's complement representation
 * for signed integer values.
 */
#if ((SCHAR_MIN + 1) != -SCHAR_MAX)
#error "This code must be compiled using a 2's complement representation for signed integer values"
#endif

/* This ID is used to detect inclusion of an incompatible rtwtypes.h */
#define RTWTYPES_ID_C08S16I32L32N32F1
#else                                  /* __TMWTYPES__ */
#define TMWTYPES_PREVIOUSLY_INCLUDED
#endif                                 /* __TMWTYPES__ */

/* Block D-Work pointer type */
typedef void * pointer_T;

/* Simulink specific types */
#ifndef __SIMSTRUC_TYPES_H__
#define __SIMSTRUC_TYPES_H__

/* Trigger directions: falling, either, and rising */
typedef enum {
  FALLING_ZERO_CROSSING = -1,
  ANY_ZERO_CROSSING = 0,
  RISING_ZERO_CROSSING = 1
} ZCDirection;

/* Previous state of a trigger signal */
typedef uint8_T ZCSigState;

/* Initial value of a trigger zero crossing signal */
#define UNINITIALIZED_ZCSIG            0x03U
#define NEG_ZCSIG                      0x02U
#define POS_ZCSIG                      0x01U
#define ZERO_ZCSIG                     0x00U

/* Current state of a trigger signal */
typedef enum {
  FALLING_ZCEVENT = -1,
  NO_ZCEVENT = 0,
  RISING_ZCEVENT = 1
} ZCEventType;

#endif                                 /* __SIMSTRUC_TYPES_H__ */
#endif                                 /* __RTWTYPES_H__ */

#ifndef MIN
#define MIN(a,b)                       ((a) < (b) ? (a) : (b))
#endif

#ifndef MAX
#define MAX(a,b)                       ((a) > (b) ? (a) : (b))
#endif
```
